PROGRAM Q4
VAR
	time_on : TIME := T#1S; 	//On for One second
	time_off : TIME := T#5S;	// Off for five seconds
	L1 : BOOL := FALSE;			// Represents the output
	TON_0: TON;
	TON_1: TON;
END_VAR

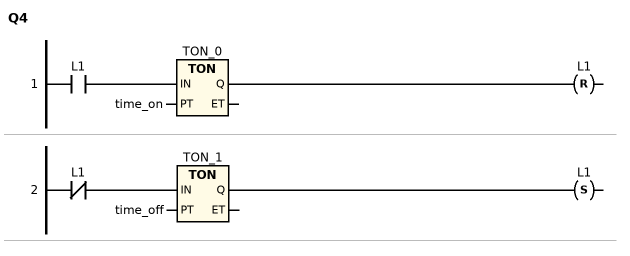
// NETWORK 1
TON_0(IN := L1, PT := time_on); // TON
L1 R= TON_0.Q;

// NETWORK 2
TON_1(IN := NOT L1, PT := time_off); // TON
L1 S= TON_1.Q;

END_PROGRAM

(* stored: Version 1.1.0.1, ProductVersion 3.1.4024.12
   POU Q4: Id {6e3285e7-69fc-432c-baeb-775a84dcb7d0}, SpecialFunc None *)
